TYPE ST_PNOutput_Battery :
STRUCT
	w_Status						:	WORD;
	w_Warnings						:	WORD;
	w_Faults						:	WORD;

	ui_SOC							: UINT;
	ui_SOH							: UINT;
	ui_DClinkVoltage 				: UINT;
	i_DClinkCurrent 				: INT;
	ui_MaxAllowedDischargeCurrent 	: UINT;
	ui_MaxAllowedChargeCurrent 		: UINT;
	i_MinCellTemperature 			: INT;
	i_MaxCellTemperature			: INT;
	ui_RemainingChargeEnergy 		: UINT;
	ui_RemainingDischargeEnergy 	: UINT;
	ui_HistAccChargeEnergy_high		: UINT;
	ui_HistAccChargeEnergy_low		: UINT;
	ui_HistAccDischargeEnergy_high	: UINT;
	ui_HistAccDischargeEnergy_low	: UINT;
END_STRUCT
END_TYPE

(* stored: Version 1.1.0.1, ProductVersion 3.1.4024.12
   DUT ST_PNOutput_Battery: Id {e85c5060-c55f-4ee4-9960-752040efbd87} *)
